FUNCTION_BLOCK CylCustom_Test EXTENDS TcUnit.FB_TestSuite IMPLEMENTS TcoCore.ITcoContext
VAR
    //Context for TcOpen
    _nfContext : TcoCore.TcoContextNfCompatibility;
END_VAR

VAR
    fbTestTimer : TON := (PT := T#30ms);
    cyl         : TcoCylinder(THIS^);
    sensor      : ARRAY[0..1] OF BOOL;
    actuator    : ARRAY[0..1] OF BOOL;
    nTestState  : INT;
END_VAR

_nfContext.VolatileOpen(); //Required for TCopen
//==============================================

ExecuteMoveToWork_SignalAtWorkShouldBeTrue();

//==============================================
_nfContext.VolatileClose();

PROPERTY Context : TcoCore.ITcoContext
GET
Context := This^._nfContext;
END_GET
END_PROPERTY

PROPERTY EndCycleCount : ULINT
GET
EndCycleCount := THIS^._nfContext._endCycleCount;
END_GET
END_PROPERTY

PROPERTY Environment : TcoCore.ITcoContextEnvironment
GET
Environment := THIS^._nfContext._settings;
END_GET
END_PROPERTY

METHOD PRIVATE ExecuteMoveToWork_SignalAtWorkShouldBeTrue
Test('ExecuteMoveToWork_SignalAtWorkShouldBeTrue');
fbTestTimer(IN := TRUE);
cyl
(
    inoAtHomePos   := sensor[0]
    , inoAtWorkPos := sensor[1]
    , inoToHomePos := actuator[0]
    , inoToWorkPos := actuator[1]
);

CASE nTestState OF
    0:
        sensor[0]  := TRUE;
        nTestState := nTestState + 1;
    1:
        // Retracted
        AssertTrue(cyl.AtHome, 'Should be AtHome');
        nTestState := nTestState + 1;
    2:
        sensor[0] := FALSE;
        cyl.MoveToWork();
        nTestState := nTestState + 1;
    3:
        AssertTrue(actuator[1], 'should turn True');
        nTestState := nTestState + 1;
    4:
        sensor[1]  := TRUE;
        nTestState := nTestState + 1;
    5:
        AssertTrue(cyl.AtWork, 'should reach Work');
END_CASE

IF fbTestTimer.Q THEN
    Assertequals_INT(Expected := 5, Actual := nTestState, Message := 'Didnt reach the last state');
    TEST_FINISHED();
END_IF
END_METHOD

PROPERTY Identity : ULINT
GET
Identity := THIS^._nfContext._Identity;
END_GET
END_PROPERTY

PROPERTY Logger : TcoCore.ITcoLogger
GET
Logger := THIS^._nfContext._logger;
END_GET
END_PROPERTY

PROPERTY RealTimeClock : TcoCore.ITcoRtc
GET
RealTimeClock := THIS^._nfContext._rtc;
END_GET
END_PROPERTY

PROPERTY StartCycleCount : ULINT
GET
StartCycleCount := THIS^._nfContext._startCycleCount;
END_GET
END_PROPERTY

END_FUNCTION_BLOCK

(* stored: Version 1.1.0.1, ProductVersion 3.1.4024.12
   POU CylCustom_Test: Id {3b4c29e4-360d-4f1b-bd78-04b5c3e6d8c7}, SpecialFunc None
   Folder ITcoContext: Id {c30550f5-1c28-485f-bff7-3d1f06f4172d}
   Property Context: Id {8d5cfcaf-62a5-48f9-8545-54f518ca6baa}
   Get Get: Id {6f448198-b903-4be2-ab39-b0580d667a78}
   Property EndCycleCount: Id {1701dea5-0b2f-4749-a493-ddd975ae114f}
   Get Get: Id {50612d92-a93c-45a5-8d3e-e29c6c0ea270}
   Property Environment: Id {1689a78d-0f9f-4e1f-9b18-95a364ab2905}
   Get Get: Id {409cd25d-54d1-49f4-96ed-a0bf49aae6c5}
   Method ExecuteMoveToWork_SignalAtWorkShouldBeTrue: Id {124bdecc-eff6-4540-89b7-1a45c3be0484}
   Property Identity: Id {e6cf42c2-97d6-4d1b-8860-590564da8696}
   Get Get: Id {e416dd72-8309-4389-9924-c10b8e7b4a0d}
   Property Logger: Id {41f32357-247c-4305-8a6f-70c03dbbf887}
   Get Get: Id {179cfd54-04d0-4bf9-90b8-1e57cf1533d7}
   Property RealTimeClock: Id {e5b28848-8d33-40e9-80fe-73d0ea6e7943}
   Get Get: Id {d6edc195-ff1c-41d0-93ea-47933d5d6a15}
   Property StartCycleCount: Id {7747fc4f-8114-4de3-a40a-fdbfa61ceed6}
   Get Get: Id {124e6984-7fc4-4eb5-8039-84014861d565} *)
